{attribute 'linkalways'}
{attribute 'hide_all_locals'}
FUNCTION_BLOCK ValueByteRead EXTENDS ValueBase IMPLEMENTS ValueRead
VAR
	thisValue : BYTE;
END_VAR

{attribute 'call_after_global_init_slot' := '1'}
{attribute 'call_after_online_change_slot' := '1'}
METHOD PROTECTED GetThisAnyType
VAR_INPUT
END_VAR
thisAnyType := ToAnyType(thisValue);
END_METHOD

METHOD GetAsType : BOOL
VAR_INPUT
	destination : __SYSTEM.AnyType;
END_VAR
GetAsType := ConvertAnyType(thisAnyType, destination);
END_METHOD

METHOD GetAsString : T_MaxString
VAR_INPUT
END_VAR
GetAsString := TO_STRING(thisValue);
END_METHOD

METHOD Get : BOOL
VAR_INPUT
	destination : ANY;
END_VAR
Get := ConvertAnyType(thisAnyType, destination);
END_METHOD

METHOD FB_init : BOOL
VAR_INPUT
	bInitRetains : BOOL; // if TRUE, the retain variables are initialized (warm start / cold start)
	bInCopyCode : BOOL;  // if TRUE, the instance afterwards gets moved into the copy code (online change)
END_VAR
_ValueType := __SYSTEM.TYPE_CLASS.TYPE_BYTE;
END_METHOD

{attribute 'monitoring' := 'call'}
PROPERTY Value : BYTE
GET
Value := thisValue;
END_GET
END_PROPERTY

END_FUNCTION_BLOCK

(* stored: Version 1.1.0.1
   POU ValueByteRead: Id {e333332e-c8c2-40c1-bb5b-e1dfd05e41ff}, SpecialFunc None
   Method GetThisAnyType: Id {3125d9ee-4add-4285-844d-5608d056d400}
   Method GetAsType: Id {3c600af1-c801-44e7-af87-04845ad73ec6}
   Method GetAsString: Id {82ed35eb-aabd-43cd-ad7e-721d44a0060e}
   Method Get: Id {9094da7e-caa6-4a92-819b-6588c93c330e}
   Method FB_init: Id {ef8abe92-1572-4c9e-8ab2-491127d5b985}
   Property Value: Id {cf36d61a-39f8-486c-abdd-c6aa30ec163a}
   Get Get: Id {c6a12bd5-0bee-4b29-9ce1-575ca29bafc5} *)
